Xinje XDPPro project, PLC1: XD5-48T6 (software 3.5.3 2018-11-19)

PROGRAM Ladder

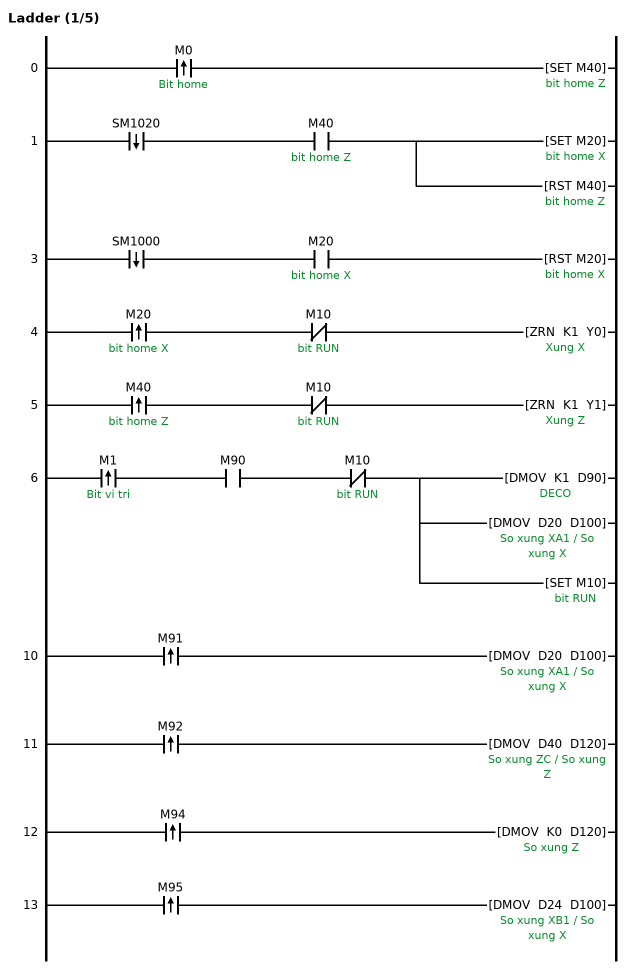
LDP    M0	; Bit home
SET    M40	; bit home Z
LDF    SM1020
AND    M40	; bit home Z
SET    M20	; bit home X
RST    M40	; bit home Z
LDF    SM1000
AND    M20	; bit home X
RST    M20	; bit home X
LDP    M20	; bit home X
ANI    M10	; bit RUN
ZRN    K1 Y0	; Xung X
LDP    M40	; bit home Z
ANI    M10	; bit RUN
ZRN    K1 Y1	; Xung Z
LDP    M1	; Bit vi tri
AND    M90
ANI    M10	; bit RUN
DMOV   K1 D90	; DECO
DMOV   D20 D100	; So xung XA1 / So xung X
SET    M10	; bit RUN
LDP    M91
DMOV   D20 D100	; So xung XA1 / So xung X
LDP    M92
DMOV   D40 D120	; So xung ZC / So xung Z
LDP    M94
DMOV   K0 D120	; So xung Z
LDP    M95
DMOV   D24 D100	; So xung XB1 / So xung X

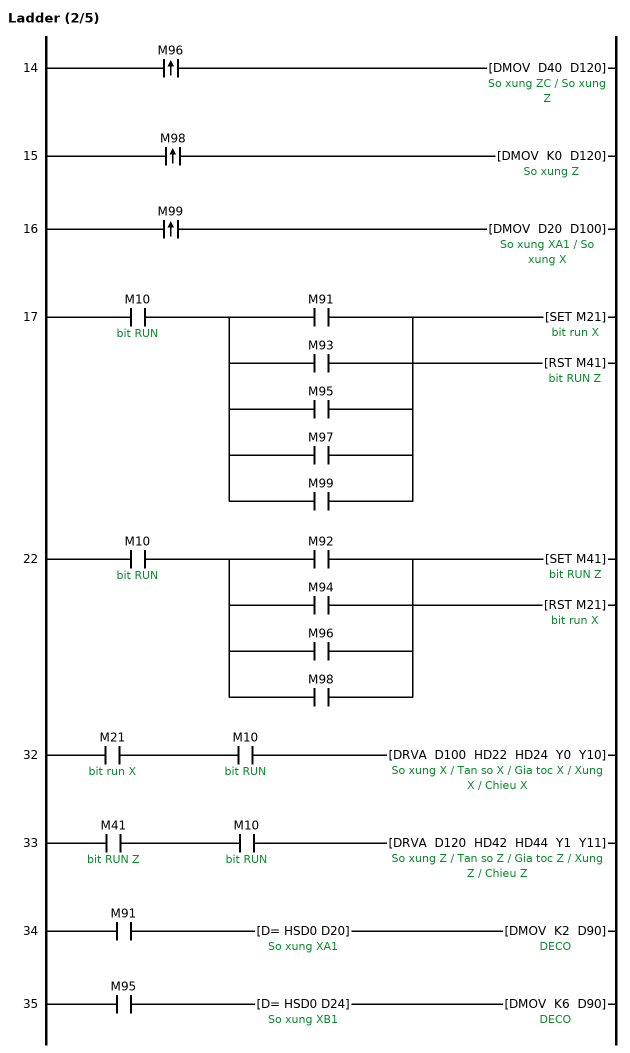
LDP    M96
DMOV   D40 D120	; So xung ZC / So xung Z
LDP    M98
DMOV   K0 D120	; So xung Z
LDP    M99
DMOV   D20 D100	; So xung XA1 / So xung X
LD     M10	; bit RUN
LD     M91
OR     M93
OR     M95
OR     M97
OR     M99
ANB
SET    M21	; bit run X
RST    M41	; bit RUN Z
LD     M10	; bit RUN
LD     M92
OR     M94
OR     M96
OR     M98
ANB
SET    M41	; bit RUN Z
RST    M21	; bit run X
LD     M21	; bit run X
AND    M10	; bit RUN
DRVA   D100 HD22 HD24 Y0 Y10	; So xung X / Tan so X / Gia toc X / Xung X / Chieu X
LD     M41	; bit RUN Z
AND    M10	; bit RUN
DRVA   D120 HD42 HD44 Y1 Y11	; So xung Z / Tan so Z / Gia toc Z / Xung Z / Chieu Z
LD     M91
DAND=  HSD0 D20	; So xung XA1
DMOV   K2 D90	; DECO
LD     M95
DAND=  HSD0 D24	; So xung XB1
DMOV   K6 D90	; DECO

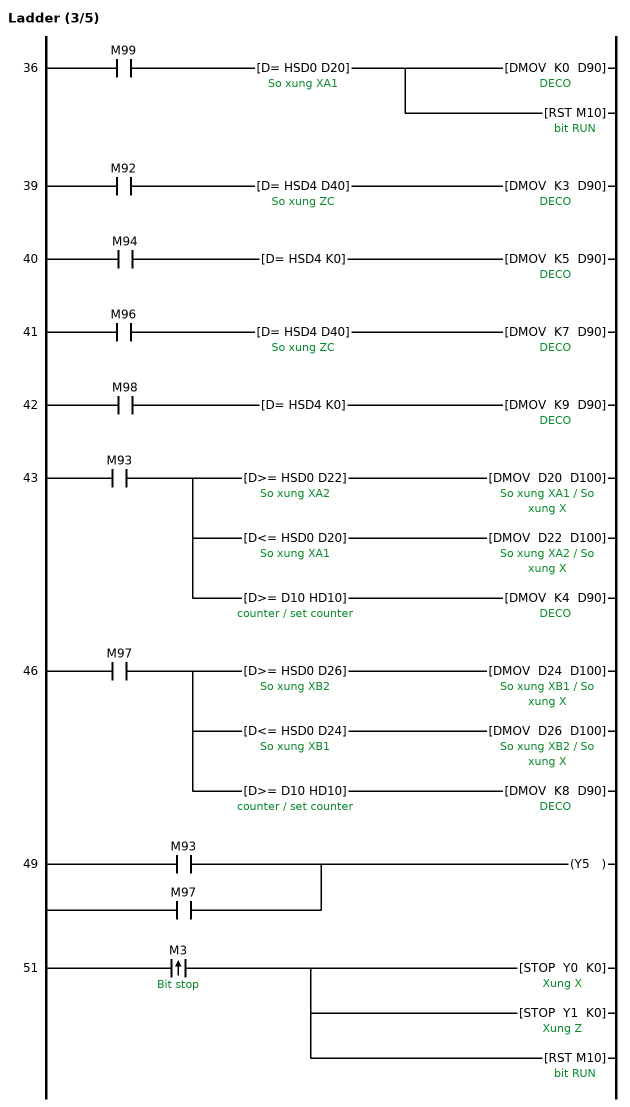
LD     M99
DAND=  HSD0 D20	; So xung XA1
DMOV   K0 D90	; DECO
RST    M10	; bit RUN
LD     M92
DAND=  HSD4 D40	; So xung ZC
DMOV   K3 D90	; DECO
LD     M94
DAND=  HSD4 K0
DMOV   K5 D90	; DECO
LD     M96
DAND=  HSD4 D40	; So xung ZC
DMOV   K7 D90	; DECO
LD     M98
DAND=  HSD4 K0
DMOV   K9 D90	; DECO
LD     M93
MPS
DAND>= HSD0 D22	; So xung XA2
DMOV   D20 D100	; So xung XA1 / So xung X
MRD
DAND<= HSD0 D20	; So xung XA1
DMOV   D22 D100	; So xung XA2 / So xung X
MPP
DAND>= D10 HD10	; counter / set counter
DMOV   K4 D90	; DECO
LD     M97
MPS
DAND>= HSD0 D26	; So xung XB2
DMOV   D24 D100	; So xung XB1 / So xung X
MRD
DAND<= HSD0 D24	; So xung XB1
DMOV   D26 D100	; So xung XB2 / So xung X
MPP
DAND>= D10 HD10	; counter / set counter
DMOV   K8 D90	; DECO
LD     M93
OR     M97
OUT    Y5
LDP    M3	; Bit stop
STOP   Y0 K0	; Xung X
STOP   Y1 K0	; Xung Z
RST    M10	; bit RUN

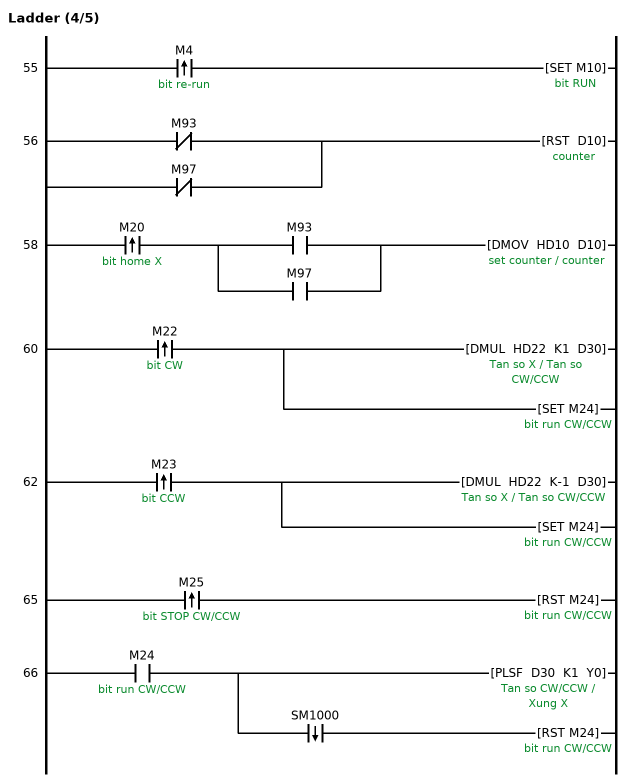
LDP    M4	; bit re-run
SET    M10	; bit RUN
LDI    M93
ORI    M97
RST    D10	; counter
LDP    M20	; bit home X
LD     M93
OR     M97
ANB
DMOV   HD10 D10	; set counter / counter
LDP    M22	; bit CW
DMUL   HD22 K1 D30	; Tan so X / Tan so CW/CCW
SET    M24	; bit run CW/CCW
LDP    M23	; bit CCW
DMUL   HD22 K-1 D30	; Tan so X / Tan so CW/CCW
SET    M24	; bit run CW/CCW
LDP    M25	; bit STOP CW/CCW
RST    M24	; bit run CW/CCW
LD     M24	; bit run CW/CCW
PLSF   D30 K1 Y0	; Tan so CW/CCW / Xung X
ANDF   SM1000
RST    M24	; bit run CW/CCW

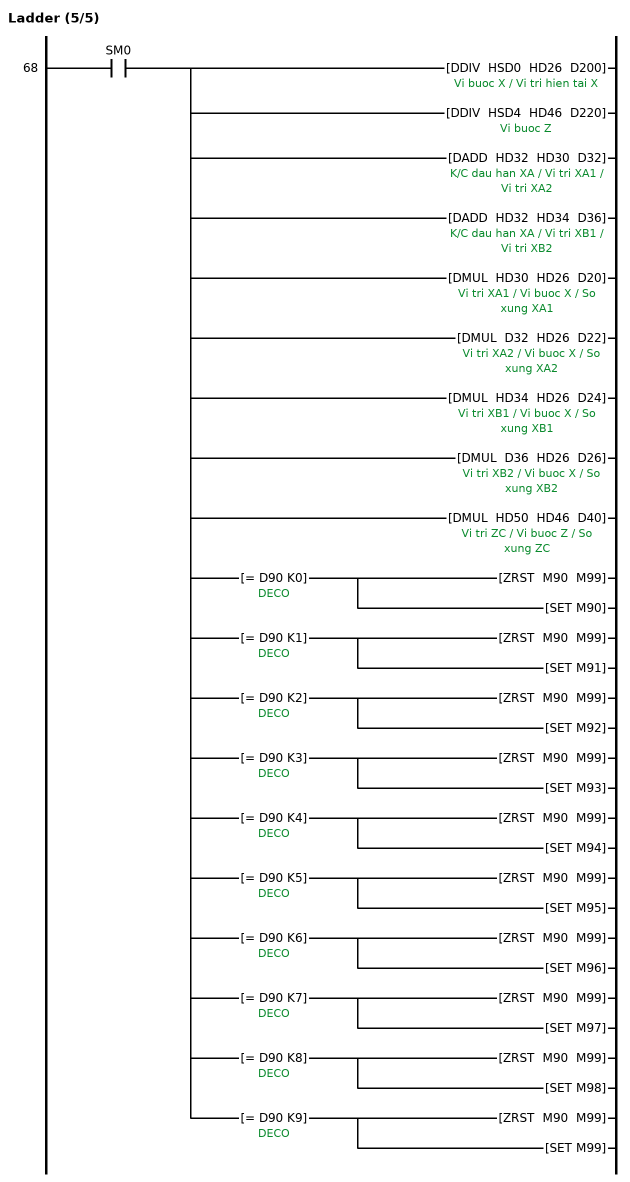
LD     SM0
DDIV   HSD0 HD26 D200	; Vi buoc X / Vi tri hien tai X
DDIV   HSD4 HD46 D220	; Vi buoc Z
DADD   HD32 HD30 D32	; K/C dau han XA / Vi tri XA1 / Vi tri XA2
DADD   HD32 HD34 D36	; K/C dau han XA / Vi tri XB1 / Vi tri XB2
DMUL   HD30 HD26 D20	; Vi tri XA1 / Vi buoc X / So xung XA1
DMUL   D32 HD26 D22	; Vi tri XA2 / Vi buoc X / So xung XA2
DMUL   HD34 HD26 D24	; Vi tri XB1 / Vi buoc X / So xung XB1
DMUL   D36 HD26 D26	; Vi tri XB2 / Vi buoc X / So xung XB2
DMUL   HD50 HD46 D40	; Vi tri ZC / Vi buoc Z / So xung ZC
MPS
AND=   D90 K0	; DECO
ZRST   M90 M99
SET    M90
MRD
AND=   D90 K1	; DECO
ZRST   M90 M99
SET    M91
MRD
AND=   D90 K2	; DECO
ZRST   M90 M99
SET    M92
MRD
AND=   D90 K3	; DECO
ZRST   M90 M99
SET    M93
MRD
AND=   D90 K4	; DECO
ZRST   M90 M99
SET    M94
MRD
AND=   D90 K5	; DECO
ZRST   M90 M99
SET    M95
MRD
AND=   D90 K6	; DECO
ZRST   M90 M99
SET    M96
MRD
AND=   D90 K7	; DECO
ZRST   M90 M99
SET    M97
MRD
AND=   D90 K8	; DECO
ZRST   M90 M99
SET    M98
MPP
AND=   D90 K9	; DECO
ZRST   M90 M99
SET    M99